FUNCTION_BLOCK LREAL_Param
VAR_INPUT PERSISTENT
	val			: LREAL;
END_VAR

END_FUNCTION_BLOCK

(* stored: Version 1.1.0.1
   POU LREAL_Param: Id {ccce5675-2e32-4b95-a41a-4221325a8283}, SpecialFunc None *)
